INTERFACE IF_Station

METHOD bearbeitenAnfordern
VAR_INPUT
	nAufnahme:		INT;
END_VAR
END_METHOD

METHOD init : BOOL
VAR_INPUT
END_VAR
END_METHOD

METHOD reset : BOOL
VAR_INPUT
END_VAR
END_METHOD

METHOD teilBearbeiten : BOOL
VAR_INPUT
END_VAR
END_METHOD

END_INTERFACE

(* stored: Version 1.1.0.1, ProductVersion 3.1.4024.12
   Itf IF_Station: Id {5667169a-38a1-45ed-af5e-430c57bf5788}
   Method bearbeitenAnfordern: Id {a689ab61-54ad-44f3-8e79-a308d6d1edd4}
   Method init: Id {a6a1835c-3dca-473a-ad94-1d32a06b7075}
   Method reset: Id {98b3e791-d6ae-4945-85f8-b61594dbb693}
   Method teilBearbeiten: Id {f0748cee-c9ee-42af-97d3-634c553a8d5a} *)
